FUNCTION WRITE_PROTECTED_STRING
VAR_INPUT
    Ptr : POINTER TO STRING;
    Value : STRING;
END_VAR

Ptr^ := Value;

END_FUNCTION

(* stored: Version 1.1.0.1, ProductVersion 3.1.4022.18
   POU WRITE_PROTECTED_STRING: Id {bad90aed-e2f4-4920-ad52-32ebaec9fc44}, SpecialFunc None *)
